// TIA Portal V19 export
DATA_BLOCK "MappedCanProcessImageOutputs"   // DB1
{ S7_Optimized_Access := 'FALSE' }
   VAR RETAIN
      statCanProcessImageOutputs { S7_SetPoint := 'True'} : "typeCanProcessImageOutputs";
   END_VAR
BEGIN
END_DATA_BLOCK
